// TIA Portal project "Assembler-Analog" (V15.1)

(* hardware
DEVICE "S7-1200 station_1"  S7-1200 Station
   slot 0: "Rack_0"  S7-1200 Rack  Rack  V1.0
   slot 1: "PLC_1"  CPU 1211C DC/DC/DC  6ES7 211-1AE40-0XB0  V4.2
DEVICE "HMI_1"  KTP900 Basic PN
   slot 0: "HMI_1"  KTP900 Basic PN  6AV2 123-2JB03-0AX0  15.1.0.0
   slot 1: "HMI_RT_1"  KTP900 Basic PN  6AV2 123-2JB03-0AX0  15.1.0.0
   slot 5: "HMI_1.IE_CP_1"  PROFINET Interface  15.0.1.0
      slot 1: "PROFINET Interface_1"  PROFINET Interface
         slot 1: "Port_1"  Port
*)

// ===== PLC "PLC_1"  CPU 1211C DC/DC/DC =====

VAR_GLOBAL   // PLC tag table "Default tag table"
   "Clock_Byte" AT %MB1869 : Byte;
   "Clock_10Hz" AT %M1869.0 : Bool;
   "Clock_5Hz" AT %M1869.1 : Bool;
   "Clock_2.5Hz" AT %M1869.2 : Bool;
   "Clock_2Hz" AT %M1869.3 : Bool;
   "Clock_1.25Hz" AT %M1869.4 : Bool;
   "Clock_1Hz" AT %M1869.5 : Bool;
   "Clock_0.625Hz" AT %M1869.6 : Bool;
   "Clock_0.5Hz" AT %M1869.7 : Bool;
   "System_Byte" AT %MB869 : Byte;
   "FirstScan" AT %M869.0 : Bool;
   "DiagStatusUpdate" AT %M869.1 : Bool;
   "AlwaysTRUE" AT %M869.2 : Bool;
   "AlwaysFALSE" AT %M869.3 : Bool;
END_VAR

VAR_GLOBAL   // PLC tag table "I/O_factory"
   "at_entry" AT %I0.0 : Bool;
   "at_entry_left" AT %I0.1 : Bool;
   "at_exit_left" AT %I0.2 : Bool;
   "at_entry_0" AT %I0.3 : Bool;
   "at_exit_0" AT %I0.4 : Bool;
   "at_entry_right" AT %I0.5 : Bool;
   "at_exit_right" AT %I0.6 : Bool;
   "at_exit" AT %I0.7 : Bool;
   "at_entry_1" AT %I1.0 : Bool;
   "at_exit_1" AT %I1.1 : Bool;
   "at_entry_2" AT %I1.2 : Bool;
   "at_exit_2" AT %I1.3 : Bool;
   "at_left_low_0" AT %I1.4 : Bool;
   "at_left_low_1" AT %I1.6 : Bool;
   "at_left_high_1" AT %I1.7 : Bool;
   "at_left_low_2" AT %I2.0 : Bool;
   "at_left_high_2" AT %I2.1 : Bool;
   "at_right_low_0" AT %I2.2 : Bool;
   "at_right_high_0" AT %I2.3 : Bool;
   "at_right_low_1" AT %I2.4 : Bool;
   "at_right_high_1" AT %I2.5 : Bool;
   "at_left_high_0" AT %I1.5 : Bool;
   "at_right_low_2" AT %I2.6 : Bool;
   "at_right_high_2" AT %I2.7 : Bool;
   "start" AT %I3.0 : Bool;
   "reset" AT %I3.1 : Bool;
   "stop" AT %I3.2 : Bool;
   "emergency_stop" AT %I3.3 : Bool;
   "auto" AT %I3.4 : Bool;
   "running" AT %I3.5 : Bool;
   "entry_conveyor" AT %Q0.0 : Bool;
   "unload_left" AT %Q0.1 : Bool;
   "load_left" AT %Q0.2 : Bool;
   "conveyor_0" AT %Q0.3 : Bool;
   "unload_right" AT %Q0.4 : Bool;
   "load_right" AT %Q0.5 : Bool;
   "exit_conveyor" AT %Q0.6 : Bool;
   "left_up" AT %Q0.7 : Bool;
   "left_slow" AT %Q1.0 : Bool;
   "left_down" AT %Q1.1 : Bool;
   "right_up" AT %Q1.2 : Bool;
   "tight_slow" AT %Q1.3 : Bool;
   "right_down" AT %Q1.4 : Bool;
   "conveyor_1" AT %Q1.5 : Bool;
   "conveyor_2" AT %Q1.6 : Bool;
   "left_warning" AT %Q1.7 : Bool;
   "right_warning" AT %Q2.0 : Bool;
   "green_0" AT %Q2.1 : Bool;
   "yellow_0" AT %Q2.2 : Bool;
   "red_0" AT %Q2.3 : Bool;
   "b_green" AT %Q2.4 : Bool;
   "b_yellow" AT %Q2.5 : Bool;
   "b_red" AT %Q2.6 : Bool;
   "c_green" AT %Q2.7 : Bool;
   "c_yellow" AT %Q3.0 : Bool;
   "c_red" AT %Q3.1 : Bool;
   "start_light" AT %Q3.2 : Bool;
   "reset_light" AT %Q3.3 : Bool;
   "stop_light" AT %Q3.4 : Bool;
END_VAR

DATA_BLOCK "Auxiliare"   // DB1
{ S7_Optimized_Access := 'TRUE' }
VERSION : 0.1
   VAR
      "counter" : DInt;
      aux_1 : Bool;
      aux_2 : Bool;
      aux_3 : Bool;
      aux_4 : Bool;
      aux_5 : Bool;
      aux_6 : Bool;
      aux_7 : Bool;
      aux_8 : Bool;
      aux_9 : Bool;
      aux_10 : Bool;
      aux_11 : Bool;
      aux_12 : Bool;
      aux_13 : Bool;
      aux_14 : Bool;
      aux_15 : Bool;
      aux_16 : Bool;
      aux_17 : Bool;
      aux_18 : Bool;
      aux_19 : Bool;
      aux_20 : Bool;
      aux_21 : Bool;
      aux_22 : Bool;
      aux_23 : Bool;
      aux_24 : Bool;
      aux_25 : Bool;
      system_stop : Bool;
   END_VAR
BEGIN
END_DATA_BLOCK

// folder: System blocks/Program resources

DATA_BLOCK "IEC_Timer_0_DB"   // DB2
{ S7_Optimized_Access := 'TRUE' }
AUTHOR : Simatic
FAMILY : IEC
NAME : IEC_TMR
VERSION : 1.0
// stored: InstanceOfName IEC_TIMER
"IEC_TIMER"
BEGIN
END_DATA_BLOCK

DATA_BLOCK "IEC_Timer_0_DB_1"   // DB4
{ S7_Optimized_Access := 'TRUE' }
AUTHOR : Simatic
FAMILY : IEC
NAME : IEC_TMR
VERSION : 1.0
// stored: InstanceOfName IEC_TIMER
"IEC_TIMER"
BEGIN
END_DATA_BLOCK

DATA_BLOCK "IEC_Timer_0_DB_2"   // DB5
{ S7_Optimized_Access := 'TRUE' }
AUTHOR : Simatic
FAMILY : IEC
NAME : IEC_TMR
VERSION : 1.0
// stored: InstanceOfName IEC_TIMER
"IEC_TIMER"
BEGIN
END_DATA_BLOCK

DATA_BLOCK "IEC_Timer_0_DB_3"   // DB6
{ S7_Optimized_Access := 'TRUE' }
AUTHOR : Simatic
FAMILY : IEC
NAME : IEC_TMR
VERSION : 1.0
// stored: InstanceOfName IEC_TIMER
"IEC_TIMER"
BEGIN
END_DATA_BLOCK

// folder: (top level)

FUNCTION "elevator" : Void   // FC1, LAD
{ S7_Optimized_Access := 'TRUE' }
VERSION : 0.1
   VAR_TEMP   // added for the SCL form of the ladder/FBD networks
      _w1 : Bool;
      _w2 : Bool;
      _w3 : Bool;
      _w4 : Bool;
      _w5 : Bool;
      _w6 : Bool;
      _w7 : Bool;
      _w8 : Bool;
      _w9 : Bool;
      _w10 : Bool;
      _w11 : Bool;
      _w12 : Bool;
      _w13 : Bool;
      _w14 : Bool;
      _w15 : Bool;
      _w16 : Bool;
      _w17 : Bool;
      _w18 : Bool;
      _w19 : Bool;
      _w20 : Bool;
   END_VAR
BEGIN

REGION Network 1: dca are conditiile de start, sa porneasca banda si lumina
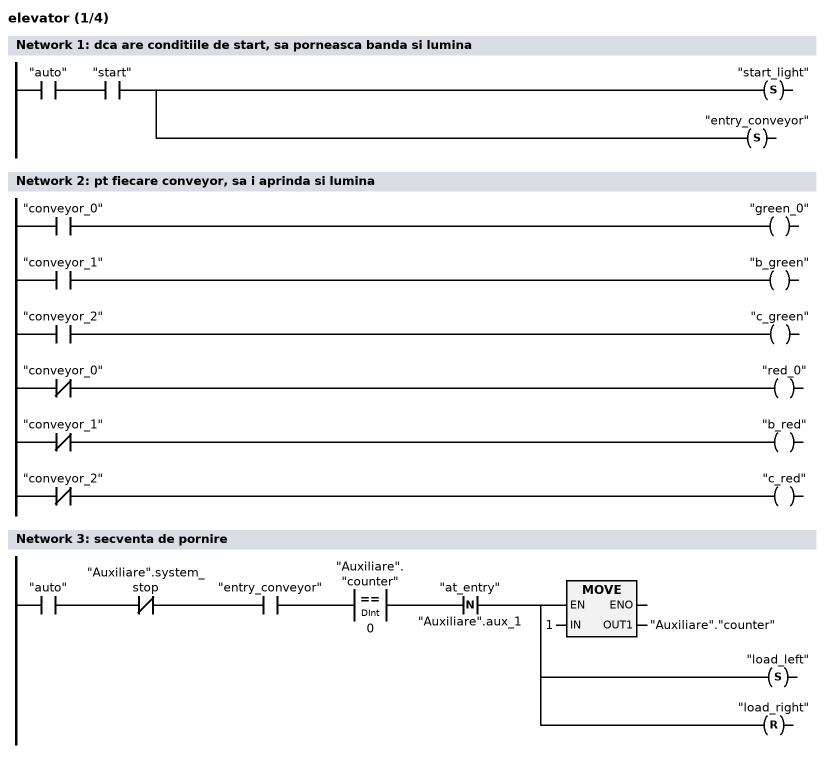
   RUNG wire#powerrail
      Contact( "auto" )
      Contact( "start" )
      wire#w1
      S_Coil( "start_light" )
   END_RUNG
   RUNG wire#w1
      S_Coil( "entry_conveyor" )
   END_RUNG
   // the same network as SCL:
   IF "auto" AND "start" THEN
       "start_light" := TRUE;
       "entry_conveyor" := TRUE;
   END_IF;
END_REGION

REGION Network 2: pt fiecare conveyor, sa i aprinda si lumina
   RUNG wire#powerrail
      Contact( "conveyor_0" )
      Coil( "green_0" )
   END_RUNG
   RUNG wire#powerrail
      Contact( "conveyor_1" )
      Coil( "b_green" )
   END_RUNG
   RUNG wire#powerrail
      Contact( "conveyor_2" )
      Coil( "c_green" )
   END_RUNG
   RUNG wire#powerrail
      I_Contact( "conveyor_0" )
      Coil( "red_0" )
   END_RUNG
   RUNG wire#powerrail
      I_Contact( "conveyor_1" )
      Coil( "b_red" )
   END_RUNG
   RUNG wire#powerrail
      I_Contact( "conveyor_2" )
      Coil( "c_red" )
   END_RUNG
   // the same network as SCL:
   "green_0" := "conveyor_0";
   "b_green" := "conveyor_1";
   "c_green" := "conveyor_2";
   "red_0" := NOT "conveyor_0";
   "b_red" := NOT "conveyor_1";
   "c_red" := NOT "conveyor_2";
END_REGION

REGION Network 3: secventa de pornire
   RUNG wire#powerrail
      Contact( "auto" )
      I_Contact( "Auxiliare".system_stop )
      Contact( "entry_conveyor" )
      { S7_Templates := "SrcType := DInt" } EQ_Contact(in1 := "Auxiliare"."counter", in2 := 0)
      N_Contact(operand := "at_entry", bit := "Auxiliare".aux_1)
      wire#w1
      Move(in := 1, out1 => "Auxiliare"."counter")
   END_RUNG
   RUNG wire#w1
      S_Coil( "load_left" )
   END_RUNG
   RUNG wire#w1
      R_Coil( "load_right" )
   END_RUNG
   // the same network as SCL:
   #_w1 := "auto" AND NOT "Auxiliare".system_stop AND "entry_conveyor" AND ("Auxiliare"."counter" = 0) AND NOT "at_entry" AND "Auxiliare".aux_1;   // falling edge of "at_entry"
   "Auxiliare".aux_1 := "at_entry";
   IF #_w1 THEN
       "Auxiliare"."counter" := 1;
       "load_left" := TRUE;
       "load_right" := FALSE;
   END_IF;
END_REGION

REGION Network 4: secvente urcari
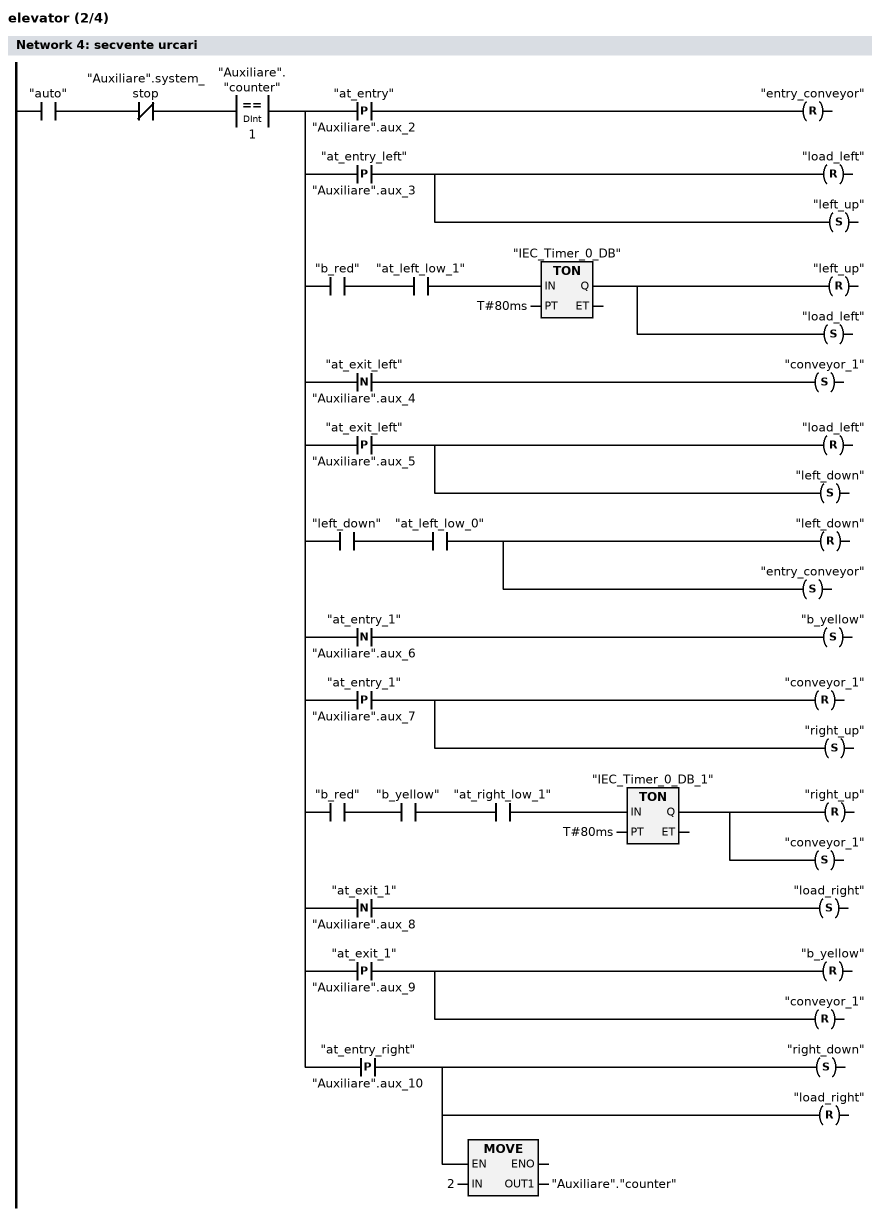
   #_w1 := "auto" AND NOT "Auxiliare".system_stop AND ("Auxiliare"."counter" = 1);
   #_w2 := #_w1 AND "at_entry" AND NOT "Auxiliare".aux_2;   // rising edge of "at_entry"
   "Auxiliare".aux_2 := "at_entry";
   IF #_w2 THEN "entry_conveyor" := FALSE; END_IF;
   #_w3 := #_w1 AND "at_entry_left" AND NOT "Auxiliare".aux_3;   // rising edge of "at_entry_left"
   "Auxiliare".aux_3 := "at_entry_left";
   IF #_w3 THEN
       "load_left" := FALSE;
       "left_up" := TRUE;
   END_IF;
   "IEC_Timer_0_DB".TON(IN := #_w1 AND "b_red" AND "at_left_low_1", PT := T#80ms);
   IF "IEC_Timer_0_DB".Q THEN
       "left_up" := FALSE;
       "load_left" := TRUE;
   END_IF;
   #_w4 := #_w1 AND NOT "at_exit_left" AND "Auxiliare".aux_4;   // falling edge of "at_exit_left"
   "Auxiliare".aux_4 := "at_exit_left";
   IF #_w4 THEN "conveyor_1" := TRUE; END_IF;
   #_w5 := #_w1 AND "at_exit_left" AND NOT "Auxiliare".aux_5;   // rising edge of "at_exit_left"
   "Auxiliare".aux_5 := "at_exit_left";
   IF #_w5 THEN
       "load_left" := FALSE;
       "left_down" := TRUE;
   END_IF;
   #_w6 := #_w1 AND "left_down" AND "at_left_low_0";
   IF #_w6 THEN
       "left_down" := FALSE;
       "entry_conveyor" := TRUE;
   END_IF;
   #_w7 := #_w1 AND NOT "at_entry_1" AND "Auxiliare".aux_6;   // falling edge of "at_entry_1"
   "Auxiliare".aux_6 := "at_entry_1";
   IF #_w7 THEN "b_yellow" := TRUE; END_IF;
   #_w8 := #_w1 AND "at_entry_1" AND NOT "Auxiliare".aux_7;   // rising edge of "at_entry_1"
   "Auxiliare".aux_7 := "at_entry_1";
   IF #_w8 THEN
       "conveyor_1" := FALSE;
       "right_up" := TRUE;
   END_IF;
   "IEC_Timer_0_DB_1".TON(IN := #_w1 AND "b_red" AND "b_yellow" AND "at_right_low_1", PT := T#80ms);
   IF "IEC_Timer_0_DB_1".Q THEN
       "right_up" := FALSE;
       "conveyor_1" := TRUE;
   END_IF;
   #_w9 := #_w1 AND NOT "at_exit_1" AND "Auxiliare".aux_8;   // falling edge of "at_exit_1"
   "Auxiliare".aux_8 := "at_exit_1";
   IF #_w9 THEN "load_right" := TRUE; END_IF;
   #_w10 := #_w1 AND "at_exit_1" AND NOT "Auxiliare".aux_9;   // rising edge of "at_exit_1"
   "Auxiliare".aux_9 := "at_exit_1";
   IF #_w10 THEN
       "b_yellow" := FALSE;
       "conveyor_1" := FALSE;
   END_IF;
   #_w11 := #_w1 AND "at_entry_right" AND NOT "Auxiliare".aux_10;   // rising edge of "at_entry_right"
   "Auxiliare".aux_10 := "at_entry_right";
   IF #_w11 THEN
       "right_down" := TRUE;
       "load_right" := FALSE;
       "Auxiliare"."counter" := 2;
   END_IF;
END_REGION

REGION Network 5: secvente coborari
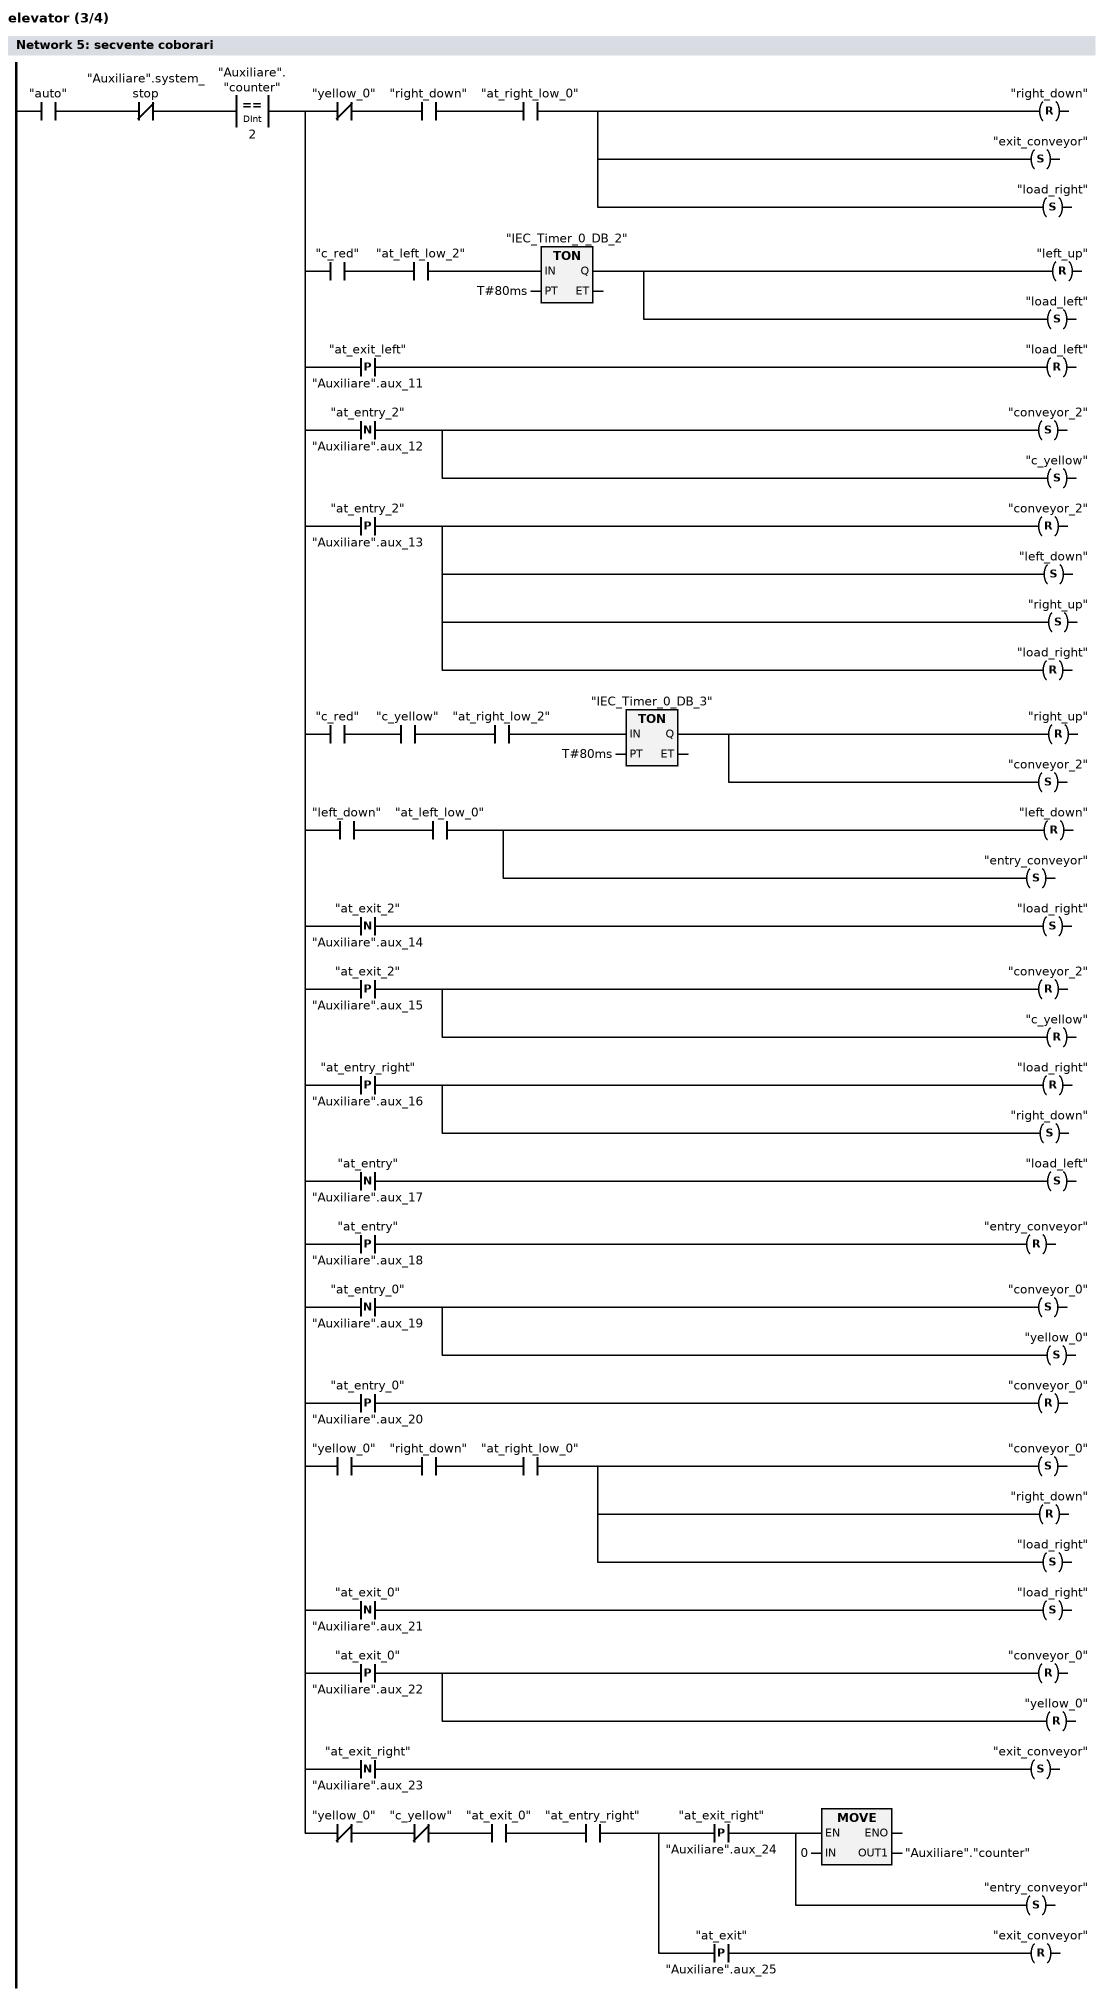
   #_w1 := "auto" AND NOT "Auxiliare".system_stop AND ("Auxiliare"."counter" = 2);
   #_w2 := #_w1 AND NOT "yellow_0" AND "right_down" AND "at_right_low_0";
   IF #_w2 THEN
       "right_down" := FALSE;
       "exit_conveyor" := TRUE;
       "load_right" := TRUE;
   END_IF;
   "IEC_Timer_0_DB_2".TON(IN := #_w1 AND "c_red" AND "at_left_low_2", PT := T#80ms);
   IF "IEC_Timer_0_DB_2".Q THEN
       "left_up" := FALSE;
       "load_left" := TRUE;
   END_IF;
   #_w3 := #_w1 AND "at_exit_left" AND NOT "Auxiliare".aux_11;   // rising edge of "at_exit_left"
   "Auxiliare".aux_11 := "at_exit_left";
   IF #_w3 THEN "load_left" := FALSE; END_IF;
   #_w4 := #_w1 AND NOT "at_entry_2" AND "Auxiliare".aux_12;   // falling edge of "at_entry_2"
   "Auxiliare".aux_12 := "at_entry_2";
   IF #_w4 THEN
       "conveyor_2" := TRUE;
       "c_yellow" := TRUE;
   END_IF;
   #_w5 := #_w1 AND "at_entry_2" AND NOT "Auxiliare".aux_13;   // rising edge of "at_entry_2"
   "Auxiliare".aux_13 := "at_entry_2";
   IF #_w5 THEN
       "conveyor_2" := FALSE;
       "left_down" := TRUE;
       "right_up" := TRUE;
       "load_right" := FALSE;
   END_IF;
   "IEC_Timer_0_DB_3".TON(IN := #_w1 AND "c_red" AND "c_yellow" AND "at_right_low_2", PT := T#80ms);
   IF "IEC_Timer_0_DB_3".Q THEN
       "right_up" := FALSE;
       "conveyor_2" := TRUE;
   END_IF;
   #_w6 := #_w1 AND "left_down" AND "at_left_low_0";
   IF #_w6 THEN
       "left_down" := FALSE;
       "entry_conveyor" := TRUE;
   END_IF;
   #_w7 := #_w1 AND NOT "at_exit_2" AND "Auxiliare".aux_14;   // falling edge of "at_exit_2"
   "Auxiliare".aux_14 := "at_exit_2";
   IF #_w7 THEN "load_right" := TRUE; END_IF;
   #_w8 := #_w1 AND "at_exit_2" AND NOT "Auxiliare".aux_15;   // rising edge of "at_exit_2"
   "Auxiliare".aux_15 := "at_exit_2";
   IF #_w8 THEN
       "conveyor_2" := FALSE;
       "c_yellow" := FALSE;
   END_IF;
   #_w9 := #_w1 AND "at_entry_right" AND NOT "Auxiliare".aux_16;   // rising edge of "at_entry_right"
   "Auxiliare".aux_16 := "at_entry_right";
   IF #_w9 THEN
       "load_right" := FALSE;
       "right_down" := TRUE;
   END_IF;
   #_w10 := #_w1 AND NOT "at_entry" AND "Auxiliare".aux_17;   // falling edge of "at_entry"
   "Auxiliare".aux_17 := "at_entry";
   IF #_w10 THEN "load_left" := TRUE; END_IF;
   #_w11 := #_w1 AND "at_entry" AND NOT "Auxiliare".aux_18;   // rising edge of "at_entry"
   "Auxiliare".aux_18 := "at_entry";
   IF #_w11 THEN "entry_conveyor" := FALSE; END_IF;
   #_w12 := #_w1 AND NOT "at_entry_0" AND "Auxiliare".aux_19;   // falling edge of "at_entry_0"
   "Auxiliare".aux_19 := "at_entry_0";
   IF #_w12 THEN
       "conveyor_0" := TRUE;
       "yellow_0" := TRUE;
   END_IF;
   #_w13 := #_w1 AND "at_entry_0" AND NOT "Auxiliare".aux_20;   // rising edge of "at_entry_0"
   "Auxiliare".aux_20 := "at_entry_0";
   IF #_w13 THEN "conveyor_0" := FALSE; END_IF;
   IF #_w1 AND "yellow_0" AND "right_down" AND "at_right_low_0" THEN "conveyor_0" := TRUE; END_IF;
   #_w14 := #_w1 AND "yellow_0" AND "right_down" AND "at_right_low_0";
   IF #_w14 THEN
       "right_down" := FALSE;
       "load_right" := TRUE;
   END_IF;
   #_w15 := #_w1 AND NOT "at_exit_0" AND "Auxiliare".aux_21;   // falling edge of "at_exit_0"
   "Auxiliare".aux_21 := "at_exit_0";
   IF #_w15 THEN "load_right" := TRUE; END_IF;
   #_w16 := #_w1 AND "at_exit_0" AND NOT "Auxiliare".aux_22;   // rising edge of "at_exit_0"
   "Auxiliare".aux_22 := "at_exit_0";
   IF #_w16 THEN
       "conveyor_0" := FALSE;
       "yellow_0" := FALSE;
   END_IF;
   #_w17 := #_w1 AND NOT "at_exit_right" AND "Auxiliare".aux_23;   // falling edge of "at_exit_right"
   "Auxiliare".aux_23 := "at_exit_right";
   IF #_w17 THEN "exit_conveyor" := TRUE; END_IF;
   #_w18 := #_w1 AND NOT "yellow_0" AND NOT "c_yellow" AND "at_exit_0" AND "at_entry_right";
   #_w19 := #_w18 AND "at_exit_right" AND NOT "Auxiliare".aux_24;   // rising edge of "at_exit_right"
   "Auxiliare".aux_24 := "at_exit_right";
   IF #_w19 THEN
       "Auxiliare"."counter" := 0;
       "entry_conveyor" := TRUE;
   END_IF;
   #_w20 := #_w18 AND "at_exit" AND NOT "Auxiliare".aux_25;   // rising edge of "at_exit"
   "Auxiliare".aux_25 := "at_exit";
   IF #_w20 THEN "exit_conveyor" := FALSE; END_IF;
END_REGION

REGION Network 6: reseteaza conditia de start
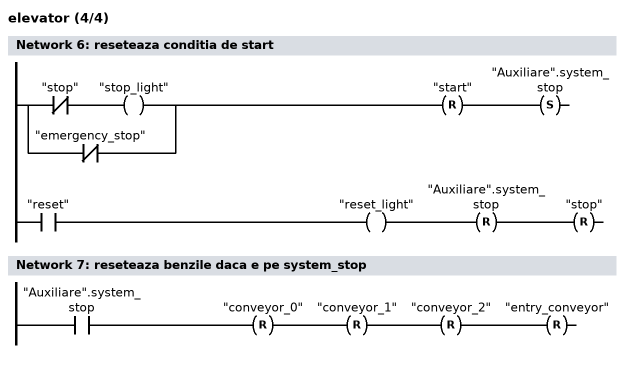
   RUNG wire#powerrail
      I_Contact( "stop" )
      Coil( "stop_light" )
      wire#w1
      R_Coil( "start" )
      S_Coil( "Auxiliare".system_stop )
   END_RUNG
   RUNG wire#powerrail
      I_Contact( "emergency_stop" )
   END_RUNG wire#w1
   RUNG wire#powerrail
      Contact( "reset" )
      Coil( "reset_light" )
      R_Coil( "Auxiliare".system_stop )
      R_Coil( "stop" )
   END_RUNG
   // the same network as SCL:
   "stop_light" := NOT "stop";
   IF NOT "stop" OR NOT "emergency_stop" THEN
       "start" := FALSE;
       "Auxiliare".system_stop := TRUE;
   END_IF;
   "reset_light" := "reset";
   IF "reset" THEN
       "Auxiliare".system_stop := FALSE;
       "stop" := FALSE;
   END_IF;
END_REGION

REGION Network 7: reseteaza benzile daca e pe system_stop
   RUNG wire#powerrail
      Contact( "Auxiliare".system_stop )
      R_Coil( "conveyor_0" )
      R_Coil( "conveyor_1" )
      R_Coil( "conveyor_2" )
      R_Coil( "entry_conveyor" )
   END_RUNG
   // the same network as SCL:
   IF "Auxiliare".system_stop THEN
       "conveyor_0" := FALSE;
       "conveyor_1" := FALSE;
       "conveyor_2" := FALSE;
       "entry_conveyor" := FALSE;
   END_IF;
END_REGION
END_FUNCTION

FUNCTION "MHJ-PLC-Lab-Function-S71200" : Void   // FC9000, SCL
{ S7_Optimized_Access := 'TRUE' }
VERSION : 0.1
   VAR_TEMP
      rdTimeReturn : Int;
      outputTime : DTL;
      SyncVal : Byte;
      forVal : Int;
      forVal_2 : Int;
      Value : Byte;
   END_VAR
   VAR CONSTANT
      CompVal : Byte := 16#34;
      Value_01 : Byte := 16#11;
      Value_01_DW : DWord := 16#A165_D992;
      Value_02_DW : DWord := 16#58BE_4401;
   END_VAR
BEGIN

   #Value:=PEEK(area := 16#82,
        dbNumber := 0,
        byteOffset := 511);
   #Value := #Value + 1;

   POKE(area := 16#82,
        dbNumber := 0,
        byteOffset := 511,
        value := #Value);

   POKE(area:=16#81,
        dbNumber:=0,
        byteOffset:=1016,
        value:=#Value_01_DW);
   POKE(area := 16#81,
        dbNumber := 0,
        byteOffset := 1020,
        value := #Value_02_DW);

   POKE(area := 16#81,
        dbNumber := 0,
        byteOffset := 511,
        value := B#16#00);

   FOR #forVal := 0 TO 120 DO
       FOR #forVal_2:=0 TO 10 DO
           #rdTimeReturn:=RD_SYS_T(#outputTime);
           #rdTimeReturn := WR_SYS_T(#outputTime);
           #rdTimeReturn := RD_SYS_T(#outputTime);
           #rdTimeReturn := WR_SYS_T(#outputTime);
       END_FOR;
       #SyncVal:= PEEK(area := 16#81,
                      dbNumber := 0,
                      byteOffset := 511);
       IF #SyncVal = #CompVal THEN
          GOTO M_1;
       END_IF;
   END_FOR;
   RETURN;

   M_1:
   POKE(area := 16#81,
        dbNumber := 0,
        byteOffset := 511,
        value := B#16#0);
END_FUNCTION

ORGANIZATION_BLOCK "Main"   // OB1, LAD, ProgramCycle
TITLE = "Main Program Sweep (Cycle)"
{ S7_Optimized_Access := 'TRUE' }
VERSION : 0.1
   VAR_INPUT
      Initial_Call : Bool;   // Initial call of this OB
      Remanence : Bool;   // =True, if remanent data are available
   END_VAR
BEGIN

REGION Network 1: fct de conectare la factory io
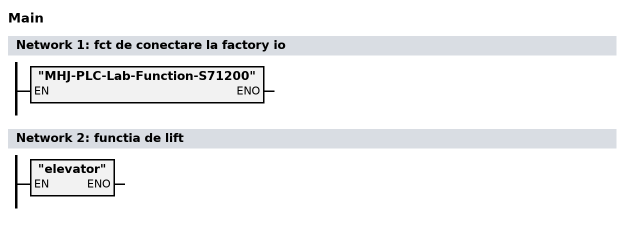
   RUNG wire#powerrail
      "MHJ-PLC-Lab-Function-S71200"()
   END_RUNG
   // the same network as SCL:
   "MHJ-PLC-Lab-Function-S71200"();
END_REGION

REGION Network 2: functia de lift
   RUNG wire#powerrail
      "elevator"()
   END_RUNG
   // the same network as SCL:
   "elevator"();
END_REGION
END_ORGANIZATION_BLOCK

(* ===== HMI "HMI_RT_1" =====
system functions are stored by id; their names below are inferred from use
connection "HMI_Connection_1": ETHERNET, SMART_S7_1200_OMS

HMI tags "Default tag table"
   "counter" : DInt = PLC counter AT %QD38, 1 s
   "Auxiliare_btn_reset_counter" : Bool = PLC Auxiliare.btn_reset_counter, 1 s
   "Alarme_gather" : Word = PLC Alarme.gather, 1 s

discrete alarms
   1: 'ESD', class Errors, trigger "Alarme_gather" bit 0

Template "Template_1" 800x480
   Button "Exit" at 722,440 size 55x39; TextOff 'Exit'; PictureOff "ExitRuntime_KTP900_Basic_PN_TR"; PictureOn "ExitRuntime_KTP900_Basic_PN_TR"
      on Release: StopRuntime(0)
   Button "Template_Button" at 622,440 size 55x39; TextOff 'Text'
   Button "Template_Button_1" at 522,440 size 55x39; TextOff 'Text'
   Button "Template_Button_2" at 422,440 size 55x39; TextOff 'Text'
   Button "Template_Button_3" at 322,440 size 55x39; TextOff 'Text'
   Button "Template_Button_4" at 222,440 size 55x39; TextOff 'Text'
   Button "Template_Button_5" at 122,440 size 55x39; TextOff 'Text'
   Button "Template_Button_6" at 22,440 size 55x39; TextOff 'Text'
*)